{attribute 'qualified_only'}
{attribute 'strict'}
TYPE E_STATES_SUPERBOHRMACHINE :
(
	initializing := 0,
	ready,
	moving,
	drilling,
	stopping,
	stopped,
	finishing
);
END_TYPE

(* stored: Version 1.1.0.1, ProductVersion 3.1.4024.3
   DUT E_STATES_SUPERBOHRMACHINE: Id {57fd385e-c900-4cb0-a10b-281833ab23e7} *)
